INTERFACE I_LogEntryAdder EXTENDS __System.IQueryInterface

METHOD AddToLogEntry : BOOL
VAR_INPUT
	refLogEntry		: REFERENCE TO FB_LogEntry;
END_VAR
END_METHOD

END_INTERFACE

(* stored: Version 1.1.0.1, ProductVersion 3.1.4024.0
   Itf I_LogEntryAdder: Id {93ca55f7-f14e-4dce-856e-2efe317067e7}
   Method AddToLogEntry: Id {667bcead-58b5-4e4b-adb9-6ccb1b9ea69e} *)
